(* PLC project PLC, Beckhoff Automation GmbH TwinCAT PLC Control 3.5.13.21 *)
(* stored: creationDateTime 2024-02-17T22:43:33.2681374, modificationDateTime 2024-02-17T22:43:33.2681374 *)

FUNCTION_BLOCK LP
VAR_INPUT
	index: LINT;
	name: STRING(G.nameStringLength);
	on: BOOL;
END_VAR
VAR_OUTPUT
END_VAR
VAR_IN_OUT
	resources: ARRAY[0..G.numAxis] OF LPResource;
END_VAR
VAR
	output: LPOutput;
	config: LPConfig;
	status: LPStatus;
END_VAR

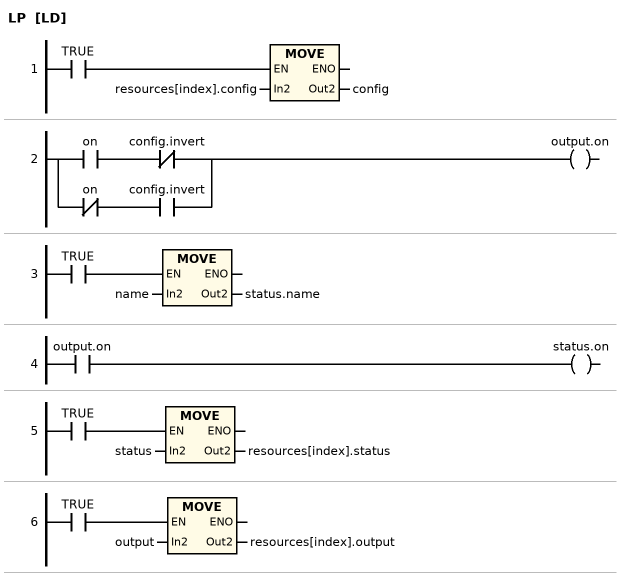
(* LD diagram, written out as Structured Text *)

IF TRUE THEN config := resources[index].config; END_IF;

output.on := on AND NOT config.invert OR NOT on AND config.invert;

IF TRUE THEN status.name := name; END_IF;

status.on := output.on;

IF TRUE THEN resources[index].status := status; END_IF;

IF TRUE THEN resources[index].output := output; END_IF;
(* --- network --- *)
END_FUNCTION_BLOCK
